FUNCTION_BLOCK EventLogger
VAR
	EventBuffer : ARRAY[1..MAXIMUM_SIZE_OF_EVENT_BUFFER] OF ST_Event;
	CurrentEventBufferIndex : INT :=0;
	
	_PersistentEventStorage : I_PersistentEventStorage;
END_VAR
VAR CONSTANT
	MAXIMUM_SIZE_OF_EVENT_BUFFER : INT := 100;
END_VAR

(* Returns TRUE if add was succesful and FALSE if buffer is full *)
METHOD PUBLIC AddEvent : BOOL
VAR_INPUT
	eEventType :E_EventType;
	eEventSeverity: Tc3_EventLogger.TcEventSeverity;
	nEventIdentity: UDINT;
	sEventText: STRING(255);
END_VAR
IF NOT IsEventBufferFull() THEN
	CurrentEventBufferIndex := CurrentEventBufferIndex + 1;
	EventBuffer[CurrentEventBufferIndex].eEventType := eEventType;
	EventBuffer[CurrentEventBufferIndex].eEventSeverity := eEventSeverity;
	EventBuffer[CurrentEventBufferIndex].nEventIdentity := nEventIdentity;
	EventBuffer[CurrentEventBufferIndex].sEventText := sEventText;
	UpdateEventTimestampWithSystemTime(stEvent := EventBuffer[CurrentEventBufferIndex]);	
//	AddEvent := TRUE;
//ELSE
//	AddEvent := FALSE;
END_IF

AddEvent := NOT IsEventBufferFull();

//Here we want to store the event persistently
_PersistentEventStorage.StoreEvent(EventBuffer[CurrentEventBufferIndex]);
END_METHOD

METHOD FB_init : BOOL
VAR_INPUT
	bInitRetains : BOOL; // if TRUE, the retain variables are initialized (warm start / cold start)
	bInCopyCode : BOOL;  // if TRUE, the instance afterwards gets moved into the copy code (online change)
	iPersistentEventStorage :I_PersistentEventStorage;
END_VAR
_PersistentEventStorage := iPersistentEventStorage;
END_METHOD

METHOD PRIVATE IsEventBufferFull : BOOL
IsEventBufferFull := (CurrentEventBufferIndex + 1) > MAXIMUM_SIZE_OF_EVENT_BUFFER;
END_METHOD

END_FUNCTION_BLOCK

(* stored: Version 1.1.0.1, ProductVersion 3.1.4024.12
   POU EventLogger: Id {009a2891-b52d-4591-8173-85c001a2e54c}, SpecialFunc None
   Method AddEvent: Id {35d26c76-d1b0-45be-9bc2-189c1f65df5c}
   Method FB_init: Id {8f538ce4-41b4-4f61-a2e1-68ea4210d3e1}
   Method IsEventBufferFull: Id {caef97e0-1154-40f2-977f-1dc855a73807} *)
